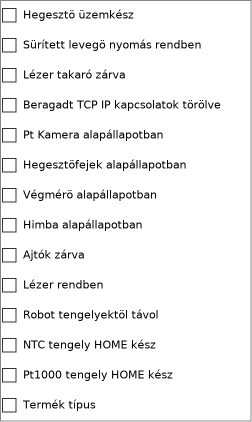
VISUALIZATION Start_ellenorzes  // 252x422
    Checkbox (0,30 250x30), "Sürített levegö nyomás rendben", variable: MAIN.bLevegoOK
    Checkbox (0,90 250x30), "Beragadt TCP IP kapcsolatok törölve", variable: INIT.bTCPKesz
    Checkbox (0,150 250x30), "Hegesztöfejek alapállapotban", variable: INIT.bHegesztoFejekKesz
    Checkbox (0,180 250x30), "Végmérö alapállapotban", variable: INIT.bVegmeroKesz
    Checkbox (0,300 250x30), "Robot tengelyektöl távol", variable: INIT.bRobotKesz
    Checkbox (0,270 250x30), "Lézer rendben", variable: INIT.bLezerKesz
    Checkbox (0,330 250x30), "NTC tengely HOME kész", variable: INIT.bNTCTengelyKesz
    Checkbox (0,360 250x30), "Pt1000 tengely HOME kész", variable: INIT.bPt1000TengelyKesz
    Checkbox (0,60 250x30), "Lézer takaró zárva", variable: VEGMERO.bLezertakaroZarva
    Checkbox (0,0 250x30), "Hegesztö üzemkész", variable: INIT.bHegesztoKesz
    Checkbox (0,390 250x30), "Termék típus", variable: GVL.bProductTypeOK
    Checkbox (0,240 250x30), "Ajtók zárva", variable: NOT GVL.bBiztonsagiFold AND GVL.bBiztonsagiTap
    Checkbox (0,210 250x30), "Himba alapállapotban", variable: INIT.bHimbaKesz
    Checkbox (0,120 250x30), "Pt Kamera alapállapotban", variable: INIT.bKameraKesz
END_VISUALIZATION

(* stored: Version 1.1.0.1, ProductVersion 3.1.4024.11
   Visu Start_ellenorzes: Id {72e7491e-d6ab-4fcd-9921-db3fcd18d37d} *)
